//{attribute 'qualified_only'}
VAR_GLOBAL
	Pendulum : Pendulum4Tc;
END_VAR

(* stored: Version 1.1.0.1, ProductVersion 3.1.4024.12
   GVL GVLPendulum: Id {e7a80d82-5e3e-4b0d-824b-96ed54cd2853} *)
